(* IEC 61131-3 sources: LTL-Test-Case-Generation/ (part 2) *)

END_FUNCTION_BLOCK

(* ---- SF_EnableSwitch2.st ---- *)
FUNCTION_BLOCK SF_EnableSwitch2
VAR_INPUT
    Activate: BOOL;
    S_SafetyActive: BOOL;
    S_EnableIn: BOOL;
    S_AutoReset: BOOL;
    Reset: BOOL;
END_VAR
VAR_OUTPUT
    Ready: BOOL;
    S_EnableSwitchOut: BOOL;
    SafetyDemand: BOOL;
    ResetRequest: BOOL;
    Error: BOOL;
    DiagCode: UINT;
END_VAR
VAR
    Reset_Before: BOOL;
END_VAR

BEGIN
// state changes

IF NOT Activate THEN
    DiagCode := 16#0000;

    Ready := FALSE;
    S_EnableSwitchOut := FALSE;
    SafetyDemand := FALSE;
    ResetRequest := FALSE;
    Error := FALSE;
    Reset_Before := FALSE;

ELSE
    IF NOT S_SafetyActive THEN
        DiagCode := 16#8002;
    ELSE
        CASE DiagCode OF
        16#0000:
            DiagCode := 16#8002;
        16#8002:
            IF (S_SafetyActive) THEN
                DiagCode := 16#8004;
            END_IF;
        16#8004:
            IF S_EnableIn THEN
                DiagCode := 16#C010;
            ELSE
                DiagCode := 16#8802;
            END_IF;
        16#8802:
            IF S_EnableIn THEN
                DiagCode := 16#8000;
            END_IF;
        16#8000:
            IF NOT S_EnableIn THEN
                DiagCode := 16#8802;
            END_IF;

        16#C010:
            IF Reset AND Reset_Before THEN
                DiagCode := 16#C011;
            ELSIF NOT S_EnableIn AND Reset AND NOT Reset_Before THEN
                DiagCode := 16#8802;
            ELSIF NOT S_EnableIn THEN
                DiagCode := 16#C410;
            END_IF;
        16#C410:
            IF Reset AND Reset_Before THEN
                DiagCode := 16#C011;
            ELSIF NOT S_EnableIn AND Reset AND NOT Reset_Before THEN
                DiagCode := 16#8802;
            ELSIF S_EnableIn THEN
                DiagCode := 16#C010;
            END_IF;
        16#C011:
            IF NOT Reset THEN
                IF S_EnableIn THEN
                    DiagCode := 16#C010;
                ELSE
                    DiagCode := 16#C410;
                END_IF;
            END_IF;
        END_CASE;
    END_IF;

    // set output variables
    CASE DiagCode OF
    16#8002:
        Ready := TRUE;
        S_EnableSwitchOut := FALSE;
        SafetyDemand := FALSE;
        ResetRequest := FALSE;
        Error := FALSE;
    16#8004:
        Ready := TRUE;
        S_EnableSwitchOut := FALSE;
        SafetyDemand := FALSE;
        ResetRequest := FALSE;
        Error := FALSE;
    16#8802:
        Ready := TRUE;
        S_EnableSwitchOut := FALSE;
        SafetyDemand := TRUE;
        ResetRequest := FALSE;
        Error := FALSE;
    16#8000:
        Ready := TRUE;
        S_EnableSwitchOut := TRUE;
        SafetyDemand := FALSE;
        ResetRequest := FALSE;
        Error := FALSE;

    // errors
    16#C011:
        Ready := TRUE;
        S_EnableSwitchOut := FALSE;
        SafetyDemand := FALSE;
        ResetRequest := FALSE;
        Error := TRUE;
    16#C010:
        Ready := TRUE;
        S_EnableSwitchOut := FALSE;
        SafetyDemand := FALSE;
        ResetRequest := FALSE;
        Error := TRUE;
    16#C410:
        Ready := TRUE;
        S_EnableSwitchOut := FALSE;
        SafetyDemand := FALSE;
        ResetRequest := NOT Reset;
        Error := TRUE;
    END_CASE;

    Reset_Before := Reset;
END_IF;

END_FUNCTION_BLOCK

(* ---- SF_EnableSwitch2_Test.st ---- *)
FUNCTION_BLOCK SF_EnableSwitch2_Test
VAR_INPUT
END_VAR
VAR_OUTPUT
	failed_0: BOOL := FALSE;
	finished_0: BOOL := FALSE;
END_VAR
VAR
	fb_0: SF_EnableSwitch2_BranchCounters;
	waitCounter_0: UINT := 0;
	testState_0: UINT := 0;
END_VAR

IF NOT failed_0 AND NOT finished_0 THEN
CASE testState_0 OF
0:
	fb_0.Activate := FALSE; fb_0.S_SafetyActive := FALSE; fb_0.S_EnableIn := FALSE; fb_0.Reset := FALSE;
	fb_0();
	failed_0 := NOT (((((((NOT (fb_0.Ready) AND NOT (fb_0.S_EnableSwitchOut)) AND NOT (fb_0.SafetyDemand)) AND NOT (fb_0.ResetRequest)) AND NOT (fb_0.Error)) AND (fb_0.DiagCode = 0)) AND NOT (fb_0.Reset_Before)));
	testState_0 := testState_0 + 1;
1:
	fb_0.Activate := TRUE; fb_0.S_SafetyActive := FALSE; fb_0.S_EnableIn := FALSE; fb_0.Reset := FALSE;
	fb_0();
	failed_0 := NOT (((((((fb_0.Ready AND NOT (fb_0.S_EnableSwitchOut)) AND NOT (fb_0.SafetyDemand)) AND NOT (fb_0.ResetRequest)) AND NOT (fb_0.Error)) AND (fb_0.DiagCode = 32770)) AND NOT (fb_0.Reset_Before)));
	testState_0 := testState_0 + 1;
2:
	fb_0.Activate := TRUE; fb_0.S_SafetyActive := FALSE; fb_0.S_EnableIn := FALSE; fb_0.Reset := FALSE;
	fb_0();
	failed_0 := NOT (((((((fb_0.Ready AND NOT (fb_0.S_EnableSwitchOut)) AND NOT (fb_0.SafetyDemand)) AND NOT (fb_0.ResetRequest)) AND NOT (fb_0.Error)) AND (fb_0.DiagCode = 32770)) AND NOT (fb_0.Reset_Before)));
	testState_0 := testState_0 + 1;
3:
	fb_0.Activate := TRUE; fb_0.S_SafetyActive := TRUE; fb_0.S_EnableIn := FALSE; fb_0.Reset := FALSE;
	fb_0();
	failed_0 := NOT (((((((fb_0.Ready AND NOT (fb_0.S_EnableSwitchOut)) AND NOT (fb_0.SafetyDemand)) AND NOT (fb_0.ResetRequest)) AND NOT (fb_0.Error)) AND (fb_0.DiagCode = 32772)) AND NOT (fb_0.Reset_Before)));
	testState_0 := testState_0 + 1;
4:
	fb_0.Activate := TRUE; fb_0.S_SafetyActive := TRUE; fb_0.S_EnableIn := FALSE; fb_0.Reset := FALSE;
	fb_0();
	failed_0 := NOT (((((((fb_0.Ready AND NOT (fb_0.S_EnableSwitchOut)) AND fb_0.SafetyDemand) AND NOT (fb_0.ResetRequest)) AND NOT (fb_0.Error)) AND (fb_0.DiagCode = 34818)) AND NOT (fb_0.Reset_Before)));
	testState_0 := testState_0 + 1;
5:
	fb_0.Activate := TRUE; fb_0.S_SafetyActive := TRUE; fb_0.S_EnableIn := FALSE; fb_0.Reset := FALSE;
	fb_0();
	failed_0 := NOT (((((((fb_0.Ready AND NOT (fb_0.S_EnableSwitchOut)) AND fb_0.SafetyDemand) AND NOT (fb_0.ResetRequest)) AND NOT (fb_0.Error)) AND (fb_0.DiagCode = 34818)) AND NOT (fb_0.Reset_Before)));
	testState_0 := testState_0 + 1;
6:
	fb_0.Activate := TRUE; fb_0.S_SafetyActive := TRUE; fb_0.S_EnableIn := TRUE; fb_0.Reset := FALSE;
	fb_0();
	failed_0 := NOT (((((((fb_0.Ready AND fb_0.S_EnableSwitchOut) AND NOT (fb_0.SafetyDemand)) AND NOT (fb_0.ResetRequest)) AND NOT (fb_0.Error)) AND (fb_0.DiagCode = 32768)) AND NOT (fb_0.Reset_Before)));
	testState_0 := testState_0 + 1;
7:
	fb_0.Activate := TRUE; fb_0.S_SafetyActive := TRUE; fb_0.S_EnableIn := TRUE; fb_0.Reset := FALSE;
	fb_0();
	failed_0 := NOT (((((((fb_0.Ready AND fb_0.S_EnableSwitchOut) AND NOT (fb_0.SafetyDemand)) AND NOT (fb_0.ResetRequest)) AND NOT (fb_0.Error)) AND (fb_0.DiagCode = 32768)) AND NOT (fb_0.Reset_Before)));
	testState_0 := testState_0 + 1;
8:
	fb_0.Activate := TRUE; fb_0.S_SafetyActive := TRUE; fb_0.S_EnableIn := FALSE; fb_0.Reset := FALSE;
	fb_0();
	failed_0 := NOT (((((((fb_0.Ready AND NOT (fb_0.S_EnableSwitchOut)) AND fb_0.SafetyDemand) AND NOT (fb_0.ResetRequest)) AND NOT (fb_0.Error)) AND (fb_0.DiagCode = 34818)) AND NOT (fb_0.Reset_Before)));
	testState_0 := testState_0 + 1;
9:
	fb_0.Activate := TRUE; fb_0.S_SafetyActive := FALSE; fb_0.S_EnableIn := FALSE; fb_0.Reset := FALSE;
	fb_0();
	failed_0 := NOT (((((((fb_0.Ready AND NOT (fb_0.S_EnableSwitchOut)) AND NOT (fb_0.SafetyDemand)) AND NOT (fb_0.ResetRequest)) AND NOT (fb_0.Error)) AND (fb_0.DiagCode = 32770)) AND NOT (fb_0.Reset_Before)));
	testState_0 := testState_0 + 1;
10:
	fb_0.Activate := TRUE; fb_0.S_SafetyActive := TRUE; fb_0.S_EnableIn := FALSE; fb_0.Reset := FALSE;
	fb_0();
	failed_0 := NOT (((((((fb_0.Ready AND NOT (fb_0.S_EnableSwitchOut)) AND NOT (fb_0.SafetyDemand)) AND NOT (fb_0.ResetRequest)) AND NOT (fb_0.Error)) AND (fb_0.DiagCode = 32772)) AND NOT (fb_0.Reset_Before)));
	testState_0 := testState_0 + 1;
11:
	fb_0.Activate := TRUE; fb_0.S_SafetyActive := TRUE; fb_0.S_EnableIn := TRUE; fb_0.Reset := TRUE;
	fb_0();
	failed_0 := NOT (((((((fb_0.Ready AND NOT (fb_0.S_EnableSwitchOut)) AND NOT (fb_0.SafetyDemand)) AND NOT (fb_0.ResetRequest)) AND fb_0.Error) AND (fb_0.DiagCode = 49168)) AND fb_0.Reset_Before));
	testState_0 := testState_0 + 1;
12:
	fb_0.Activate := TRUE; fb_0.S_SafetyActive := TRUE; fb_0.S_EnableIn := TRUE; fb_0.Reset := TRUE;
	fb_0();
	failed_0 := NOT (((((((fb_0.Ready AND NOT (fb_0.S_EnableSwitchOut)) AND NOT (fb_0.SafetyDemand)) AND NOT (fb_0.ResetRequest)) AND fb_0.Error) AND (fb_0.DiagCode = 49169)) AND fb_0.Reset_Before));
	testState_0 := testState_0 + 1;
13:
	fb_0.Activate := TRUE; fb_0.S_SafetyActive := TRUE; fb_0.S_EnableIn := TRUE; fb_0.Reset := TRUE;
	fb_0();
	failed_0 := NOT (((((((fb_0.Ready AND NOT (fb_0.S_EnableSwitchOut)) AND NOT (fb_0.SafetyDemand)) AND NOT (fb_0.ResetRequest)) AND fb_0.Error) AND (fb_0.DiagCode = 49169)) AND fb_0.Reset_Before));
	testState_0 := testState_0 + 1;
14:
	fb_0.Activate := TRUE; fb_0.S_SafetyActive := TRUE; fb_0.S_EnableIn := TRUE; fb_0.Reset := FALSE;
	fb_0();
	failed_0 := NOT (((((((fb_0.Ready AND NOT (fb_0.S_EnableSwitchOut)) AND NOT (fb_0.SafetyDemand)) AND NOT (fb_0.ResetRequest)) AND fb_0.Error) AND (fb_0.DiagCode = 49168)) AND NOT (fb_0.Reset_Before)));
	testState_0 := testState_0 + 1;
15:
	fb_0.Activate := TRUE; fb_0.S_SafetyActive := TRUE; fb_0.S_EnableIn := TRUE; fb_0.Reset := FALSE;
	fb_0();
	failed_0 := NOT (((((((fb_0.Ready AND NOT (fb_0.S_EnableSwitchOut)) AND NOT (fb_0.SafetyDemand)) AND NOT (fb_0.ResetRequest)) AND fb_0.Error) AND (fb_0.DiagCode = 49168)) AND NOT (fb_0.Reset_Before)));
	testState_0 := testState_0 + 1;
16:
	fb_0.Activate := TRUE; fb_0.S_SafetyActive := TRUE; fb_0.S_EnableIn := FALSE; fb_0.Reset := FALSE;
	fb_0();
	failed_0 := NOT (((((((fb_0.Ready AND NOT (fb_0.S_EnableSwitchOut)) AND NOT (fb_0.SafetyDemand)) AND fb_0.ResetRequest) AND fb_0.Error) AND (fb_0.DiagCode = 50192)) AND NOT (fb_0.Reset_Before)));
	testState_0 := testState_0 + 1;
17:
	fb_0.Activate := TRUE; fb_0.S_SafetyActive := TRUE; fb_0.S_EnableIn := FALSE; fb_0.Reset := FALSE;
	fb_0();
	failed_0 := NOT (((((((fb_0.Ready AND NOT (fb_0.S_EnableSwitchOut)) AND NOT (fb_0.SafetyDemand)) AND fb_0.ResetRequest) AND fb_0.Error) AND (fb_0.DiagCode = 50192)) AND NOT (fb_0.Reset_Before)));
	testState_0 := testState_0 + 1;
18:
	fb_0.Activate := TRUE; fb_0.S_SafetyActive := TRUE; fb_0.S_EnableIn := TRUE; fb_0.Reset := FALSE;
	fb_0();
	failed_0 := NOT (((((((fb_0.Ready AND NOT (fb_0.S_EnableSwitchOut)) AND NOT (fb_0.SafetyDemand)) AND NOT (fb_0.ResetRequest)) AND fb_0.Error) AND (fb_0.DiagCode = 49168)) AND NOT (fb_0.Reset_Before)));
	testState_0 := testState_0 + 1;
19:
	fb_0.Activate := TRUE; fb_0.S_SafetyActive := TRUE; fb_0.S_EnableIn := FALSE; fb_0.Reset := TRUE;
	fb_0();
	failed_0 := NOT (((((((fb_0.Ready AND NOT (fb_0.S_EnableSwitchOut)) AND fb_0.SafetyDemand) AND NOT (fb_0.ResetRequest)) AND NOT (fb_0.Error)) AND (fb_0.DiagCode = 34818)) AND fb_0.Reset_Before));
	testState_0 := testState_0 + 1;
20:
	fb_0.Activate := TRUE; fb_0.S_SafetyActive := FALSE; fb_0.S_EnableIn := FALSE; fb_0.Reset := FALSE;
	fb_0();
	failed_0 := NOT (((((((fb_0.Ready AND NOT (fb_0.S_EnableSwitchOut)) AND NOT (fb_0.SafetyDemand)) AND NOT (fb_0.ResetRequest)) AND NOT (fb_0.Error)) AND (fb_0.DiagCode = 32770)) AND NOT (fb_0.Reset_Before)));
	testState_0 := testState_0 + 1;
21:
	fb_0.Activate := TRUE; fb_0.S_SafetyActive := FALSE; fb_0.S_EnableIn := FALSE; fb_0.Reset := FALSE;
	fb_0();
	failed_0 := NOT (((((((fb_0.Ready AND NOT (fb_0.S_EnableSwitchOut)) AND NOT (fb_0.SafetyDemand)) AND NOT (fb_0.ResetRequest)) AND NOT (fb_0.Error)) AND (fb_0.DiagCode = 32770)) AND NOT (fb_0.Reset_Before)));
	testState_0 := testState_0 + 1;
22:
	fb_0.Activate := TRUE; fb_0.S_SafetyActive := TRUE; fb_0.S_EnableIn := FALSE; fb_0.Reset := FALSE;
	fb_0();
	failed_0 := NOT (((((((fb_0.Ready AND NOT (fb_0.S_EnableSwitchOut)) AND NOT (fb_0.SafetyDemand)) AND NOT (fb_0.ResetRequest)) AND NOT (fb_0.Error)) AND (fb_0.DiagCode = 32772)) AND NOT (fb_0.Reset_Before)));
	testState_0 := testState_0 + 1;
23:
	fb_0.Activate := TRUE; fb_0.S_SafetyActive := TRUE; fb_0.S_EnableIn := TRUE; fb_0.Reset := TRUE;
	fb_0();
	failed_0 := NOT (((((((fb_0.Ready AND NOT (fb_0.S_EnableSwitchOut)) AND NOT (fb_0.SafetyDemand)) AND NOT (fb_0.ResetRequest)) AND fb_0.Error) AND (fb_0.DiagCode = 49168)) AND fb_0.Reset_Before));
	testState_0 := testState_0 + 1;
24:
	fb_0.Activate := TRUE; fb_0.S_SafetyActive := TRUE; fb_0.S_EnableIn := FALSE; fb_0.Reset := TRUE;
	fb_0();
	failed_0 := NOT (((((((fb_0.Ready AND NOT (fb_0.S_EnableSwitchOut)) AND NOT (fb_0.SafetyDemand)) AND NOT (fb_0.ResetRequest)) AND fb_0.Error) AND (fb_0.DiagCode = 49169)) AND fb_0.Reset_Before));
	testState_0 := testState_0 + 1;
25:
	fb_0.Activate := TRUE; fb_0.S_SafetyActive := TRUE; fb_0.S_EnableIn := FALSE; fb_0.Reset := FALSE;
	fb_0();
	failed_0 := NOT (((((((fb_0.Ready AND NOT (fb_0.S_EnableSwitchOut)) AND NOT (fb_0.SafetyDemand)) AND fb_0.ResetRequest) AND fb_0.Error) AND (fb_0.DiagCode = 50192)) AND NOT (fb_0.Reset_Before)));
	testState_0 := testState_0 + 1;
26:
	fb_0.Activate := TRUE; fb_0.S_SafetyActive := TRUE; fb_0.S_EnableIn := FALSE; fb_0.Reset := TRUE;
	fb_0();
	failed_0 := NOT (((((((fb_0.Ready AND NOT (fb_0.S_EnableSwitchOut)) AND fb_0.SafetyDemand) AND NOT (fb_0.ResetRequest)) AND NOT (fb_0.Error)) AND (fb_0.DiagCode = 34818)) AND fb_0.Reset_Before));
	testState_0 := testState_0 + 1;
27:
	fb_0.Activate := TRUE; fb_0.S_SafetyActive := FALSE; fb_0.S_EnableIn := FALSE; fb_0.Reset := FALSE;
	fb_0();
	failed_0 := NOT ((fb_0.Ready AND (NOT (fb_0.S_EnableSwitchOut) AND (NOT (fb_0.SafetyDemand) AND (NOT (fb_0.ResetRequest) AND (NOT (fb_0.Error) AND ((fb_0.DiagCode = 32770) AND NOT (fb_0.Reset_Before))))))));
	testState_0 := testState_0 + 1;
28:
	finished_0 := TRUE;
END_CASE
END_IF

END_FUNCTION_BLOCK

(* ---- SF_Equivalent_U.st ---- *)
FUNCTION_BLOCK SF_Equivalent_U
VAR_INPUT
    Activate: BOOL;
    S_ChannelA: BOOL;
    S_ChannelB: BOOL;
    DiscrepancyTime: TIME := T#100ms;
END_VAR
VAR_OUTPUT
    Ready: BOOL;
    S_EquivalentOut: BOOL;
    SafetyDemand: BOOL;
    Error: BOOL;
    DiagCode: UINT;
END_VAR
VAR
    T_1: TON;
END_VAR

BEGIN

// state changes
IF NOT Activate THEN
    DiagCode := 16#0000;
    T_1(IN := 0);

    Ready := FALSE;
    SafetyDemand := FALSE;
    Error := FALSE;
    S_EquivalentOut := FALSE;
ELSE
    T_1(PT := DiscrepancyTime);

    CASE DiagCode OF
    16#0000:
        DiagCode := 16#8801;
    16#8000:
        IF S_ChannelA XOR S_ChannelB THEN
            DiagCode := 16#8806;
            T_1(IN := 0);
            T_1(IN := 1, PT := DiscrepancyTime);
        ELSIF NOT S_ChannelA AND NOT S_ChannelB THEN
            T_1(IN := 0);
            DiagCode := 16#8801;
        END_IF;
    16#8801:
        IF S_ChannelA AND NOT S_ChannelB THEN
            DiagCode := 16#8802;
            T_1(IN := 0);
            T_1(IN := 1, PT := DiscrepancyTime);
        ELSIF S_ChannelB AND NOT S_ChannelA THEN
            DiagCode := 16#8804;
            T_1(IN := 0);
            T_1(IN := 1, PT := DiscrepancyTime);
        ELSIF S_ChannelA AND S_ChannelB THEN
            DiagCode := 16#8000;
        END_IF;
    16#8802:
        IF T_1.Q THEN
            DiagCode := 16#C010;
        ELSIF NOT S_ChannelA THEN
            T_1(IN := 0);
            DiagCode := 16#8801;
        ELSIF S_ChannelB THEN
            T_1(IN := 0);
            DiagCode := 16#8000;
        END_IF;
    16#8804:
        IF T_1.Q THEN
            DiagCode := 16#C020;
        ELSIF NOT S_ChannelB THEN
            T_1(IN := 0);
            DiagCode := 16#8801;
        ELSIF S_ChannelA THEN
            T_1(IN := 0);
            DiagCode := 16#8000;
        END_IF;
    16#8806:
        IF T_1.Q THEN
            DiagCode := 16#C030;
        ELSIF NOT S_ChannelA AND NOT S_ChannelB THEN
            T_1(IN := 0);
            DiagCode := 16#8801;
        END_IF;
    16#C010:
        IF NOT S_ChannelA AND NOT S_ChannelB THEN
            T_1(IN := 0);
            DiagCode := 16#8801;
        END_IF;
    16#C020:
        IF NOT S_ChannelA AND NOT S_ChannelB THEN
            T_1(IN := 0);
            DiagCode := 16#8801;
        END_IF;
    16#C030:
        IF NOT S_ChannelA AND NOT S_ChannelB THEN
            T_1(IN := 0);
            DiagCode := 16#8801;
        END_IF;
    END_CASE;

    // set output variables
    CASE DiagCode OF
    16#8000:
        Ready := TRUE;
        SafetyDemand := FALSE;
        Error := FALSE;
        S_EquivalentOut := TRUE;
    16#8801:
        Ready := TRUE;
        SafetyDemand := TRUE;
        Error := FALSE;
        S_EquivalentOut := FALSE;
    16#8802:
        Ready := TRUE;
        SafetyDemand := TRUE;
        Error := FALSE;
        S_EquivalentOut := FALSE;
    16#8804:
        Ready := TRUE;
        SafetyDemand := TRUE;
        Error := FALSE;
        S_EquivalentOut := FALSE;
    16#8806:
        Ready := TRUE;
        SafetyDemand := TRUE;
        Error := FALSE;
        S_EquivalentOut := FALSE;
    16#C010:
        Ready := TRUE;
        SafetyDemand := FALSE;
        Error := TRUE;
        S_EquivalentOut := FALSE;
    16#C020:
        Ready := TRUE;
        SafetyDemand := FALSE;
        Error := TRUE;
        S_EquivalentOut := FALSE;
    16#C030:
        Ready := TRUE;
        SafetyDemand := FALSE;
        Error := TRUE;
        S_EquivalentOut := FALSE;
    END_CASE;
END_IF;

END_FUNCTION_BLOCK

(* ---- SF_Equivalent_U_Test.st ---- *)
FUNCTION_BLOCK SF_Equivalent_U_Test
VAR_INPUT
END_VAR
VAR_OUTPUT
	failed_0: BOOL := FALSE;
	finished_0: BOOL := FALSE;
END_VAR
VAR
	fb_0: SF_Equivalent_U_BranchCounters;
	waitCounter_0: UINT := 0;
	testState_0: UINT := 0;
END_VAR

IF NOT failed_0 AND NOT finished_0 THEN
CASE testState_0 OF
0:
	fb_0.Activate := FALSE;
	fb_0();
	failed_0 := NOT ((((((NOT (fb_0.T_1.Q) AND (fb_0.DiagCode = 0)) AND NOT (fb_0.Ready)) AND NOT (fb_0.S_EquivalentOut)) AND NOT (fb_0.SafetyDemand)) AND NOT (fb_0.Error)));
	testState_0 := testState_0 + 1;
1:
	fb_0.Activate := TRUE; fb_0.S_ChannelA := FALSE; fb_0.S_ChannelB := FALSE;
	fb_0();
	failed_0 := NOT ((((((NOT (fb_0.T_1.Q) AND (fb_0.DiagCode = 34817)) AND fb_0.Ready) AND NOT (fb_0.S_EquivalentOut)) AND fb_0.SafetyDemand) AND NOT (fb_0.Error)));
	testState_0 := testState_0 + 1;
2:
	fb_0.Activate := TRUE; fb_0.S_ChannelA := FALSE; fb_0.S_ChannelB := FALSE;
	fb_0();
	failed_0 := NOT ((((((NOT (fb_0.T_1.Q) AND (fb_0.DiagCode = 34817)) AND fb_0.Ready) AND NOT (fb_0.S_EquivalentOut)) AND fb_0.SafetyDemand) AND NOT (fb_0.Error)));
	testState_0 := testState_0 + 1;
3:
	fb_0.Activate := TRUE; fb_0.S_ChannelA := TRUE; fb_0.S_ChannelB := FALSE;
	fb_0();
	failed_0 := NOT ((((((NOT (fb_0.T_1.Q) AND (fb_0.DiagCode = 34818)) AND fb_0.Ready) AND NOT (fb_0.S_EquivalentOut)) AND fb_0.SafetyDemand) AND NOT (fb_0.Error)));
	testState_0 := testState_0 + 1;
4:
	fb_0.Activate := TRUE; fb_0.S_ChannelA := FALSE; fb_0.S_ChannelB := FALSE;
	fb_0();
	IF fb_0.T_1.Q THEN
		finished_0 := TRUE;
	ELSE
		testState_0 := testState_0 + 1;
	END_IF
5:
	failed_0 := NOT ((((((NOT (fb_0.T_1.Q) AND (fb_0.DiagCode = 34817)) AND fb_0.Ready) AND NOT (fb_0.S_EquivalentOut)) AND fb_0.SafetyDemand) AND NOT (fb_0.Error)));
	testState_0 := testState_0 + 1;
6:
	fb_0.Activate := TRUE; fb_0.S_ChannelA := TRUE; fb_0.S_ChannelB := FALSE;
	fb_0();
	failed_0 := NOT ((((((NOT (fb_0.T_1.Q) AND (fb_0.DiagCode = 34818)) AND fb_0.Ready) AND NOT (fb_0.S_EquivalentOut)) AND fb_0.SafetyDemand) AND NOT (fb_0.Error)));
	testState_0 := testState_0 + 1;
7:
	fb_0.Activate := TRUE; fb_0.S_ChannelA := TRUE; fb_0.S_ChannelB := TRUE;
	fb_0();
	IF fb_0.T_1.Q THEN
		finished_0 := TRUE;
	ELSE
		testState_0 := testState_0 + 1;
	END_IF
8:
	failed_0 := NOT ((((((NOT (fb_0.T_1.Q) AND (fb_0.DiagCode = 32768)) AND fb_0.Ready) AND fb_0.S_EquivalentOut) AND NOT (fb_0.SafetyDemand)) AND NOT (fb_0.Error)));
	testState_0 := testState_0 + 1;
9:
	fb_0.Activate := TRUE; fb_0.S_ChannelA := TRUE; fb_0.S_ChannelB := TRUE;
	fb_0();
	failed_0 := NOT ((((((NOT (fb_0.T_1.Q) AND (fb_0.DiagCode = 32768)) AND fb_0.Ready) AND fb_0.S_EquivalentOut) AND NOT (fb_0.SafetyDemand)) AND NOT (fb_0.Error)));
	testState_0 := testState_0 + 1;
10:
	fb_0.Activate := TRUE; fb_0.S_ChannelA := FALSE; fb_0.S_ChannelB := TRUE;
	fb_0();
	failed_0 := NOT ((((((NOT (fb_0.T_1.Q) AND (fb_0.DiagCode = 34822)) AND fb_0.Ready) AND NOT (fb_0.S_EquivalentOut)) AND fb_0.SafetyDemand) AND NOT (fb_0.Error)));
	testState_0 := testState_0 + 1;
11:
	fb_0.Activate := TRUE; fb_0.S_ChannelA := FALSE; fb_0.S_ChannelB := FALSE;
	fb_0();
	IF fb_0.T_1.Q THEN
		finished_0 := TRUE;
	ELSE
		testState_0 := testState_0 + 1;
	END_IF
12:
	failed_0 := NOT ((((((NOT (fb_0.T_1.Q) AND (fb_0.DiagCode = 34817)) AND fb_0.Ready) AND NOT (fb_0.S_EquivalentOut)) AND fb_0.SafetyDemand) AND NOT (fb_0.Error)));
	testState_0 := testState_0 + 1;
13:
	fb_0.Activate := TRUE; fb_0.S_ChannelA := FALSE; fb_0.S_ChannelB := TRUE;
	fb_0();
	failed_0 := NOT ((((((NOT (fb_0.T_1.Q) AND (fb_0.DiagCode = 34820)) AND fb_0.Ready) AND NOT (fb_0.S_EquivalentOut)) AND fb_0.SafetyDemand) AND NOT (fb_0.Error)));
	testState_0 := testState_0 + 1;
14:
	fb_0.Activate := TRUE; fb_0.S_ChannelA := FALSE; fb_0.S_ChannelB := FALSE;
	fb_0();
	IF fb_0.T_1.Q THEN
		finished_0 := TRUE;
	ELSE
		testState_0 := testState_0 + 1;
	END_IF
15:
	failed_0 := NOT ((((((NOT (fb_0.T_1.Q) AND (fb_0.DiagCode = 34817)) AND fb_0.Ready) AND NOT (fb_0.S_EquivalentOut)) AND fb_0.SafetyDemand) AND NOT (fb_0.Error)));
	testState_0 := testState_0 + 1;
16:
	fb_0.Activate := TRUE; fb_0.S_ChannelA := FALSE; fb_0.S_ChannelB := TRUE;
	fb_0();
	failed_0 := NOT ((((((NOT (fb_0.T_1.Q) AND (fb_0.DiagCode = 34820)) AND fb_0.Ready) AND NOT (fb_0.S_EquivalentOut)) AND fb_0.SafetyDemand) AND NOT (fb_0.Error)));
	testState_0 := testState_0 + 1;
17:
	fb_0.Activate := TRUE; fb_0.S_ChannelA := TRUE; fb_0.S_ChannelB := TRUE;
	fb_0();
	IF fb_0.T_1.Q THEN
		finished_0 := TRUE;
	ELSE
		testState_0 := testState_0 + 1;
	END_IF
18:
	failed_0 := NOT ((((((NOT (fb_0.T_1.Q) AND (fb_0.DiagCode = 32768)) AND fb_0.Ready) AND fb_0.S_EquivalentOut) AND NOT (fb_0.SafetyDemand)) AND NOT (fb_0.Error)));
	testState_0 := testState_0 + 1;
19:
	fb_0.Activate := TRUE; fb_0.S_ChannelA := FALSE; fb_0.S_ChannelB := FALSE;
	fb_0();
	failed_0 := NOT ((((((NOT (fb_0.T_1.Q) AND (fb_0.DiagCode = 34817)) AND fb_0.Ready) AND NOT (fb_0.S_EquivalentOut)) AND fb_0.SafetyDemand) AND NOT (fb_0.Error)));
	testState_0 := testState_0 + 1;
20:
	fb_0.Activate := TRUE; fb_0.S_ChannelA := TRUE; fb_0.S_ChannelB := TRUE;
	fb_0();
	failed_0 := NOT ((((((NOT (fb_0.T_1.Q) AND (fb_0.DiagCode = 32768)) AND fb_0.Ready) AND fb_0.S_EquivalentOut) AND NOT (fb_0.SafetyDemand)) AND NOT (fb_0.Error)));
	testState_0 := testState_0 + 1;
21:
	fb_0.Activate := TRUE; fb_0.S_ChannelA := TRUE; fb_0.S_ChannelB := FALSE;
	fb_0();
	failed_0 := NOT ((((((NOT (fb_0.T_1.Q) AND (fb_0.DiagCode = 34822)) AND fb_0.Ready) AND NOT (fb_0.S_EquivalentOut)) AND fb_0.SafetyDemand) AND NOT (fb_0.Error)));
	testState_0 := testState_0 + 1;
22:
	IF (fb_0.T_1.Q AND (fb_0.DiagCode = 49200)) THEN
		waitCounter_0 := 0;
		testState_0 := testState_0 + 1;
	ELSE
		failed_0 := NOT ((NOT (fb_0.T_1.Q) AND ((fb_0.DiagCode = 34822) AND (fb_0.Ready AND (NOT (fb_0.S_EquivalentOut) AND (fb_0.SafetyDemand AND NOT (fb_0.Error)))))));
		IF waitCounter_0 > 100 THEN
			finished_0 := TRUE;
		ELSE
			waitCounter_0 := waitCounter_0 + 1;
			fb_0();
		END_IF
	END_IF
23:
	failed_0 := NOT ((((((fb_0.T_1.Q AND (fb_0.DiagCode = 49200)) AND fb_0.Ready) AND NOT (fb_0.S_EquivalentOut)) AND NOT (fb_0.SafetyDemand)) AND fb_0.Error));
	testState_0 := testState_0 + 1;
24:
	fb_0.Activate := TRUE; fb_0.S_ChannelA := TRUE; fb_0.S_ChannelB := FALSE;
	fb_0();
	failed_0 := NOT ((((((fb_0.T_1.Q AND (fb_0.DiagCode = 49200)) AND fb_0.Ready) AND NOT (fb_0.S_EquivalentOut)) AND NOT (fb_0.SafetyDemand)) AND fb_0.Error));
	testState_0 := testState_0 + 1;
25:
	fb_0.Activate := TRUE; fb_0.S_ChannelA := FALSE; fb_0.S_ChannelB := FALSE;
	fb_0();
	failed_0 := NOT ((((((NOT (fb_0.T_1.Q) AND (fb_0.DiagCode = 34817)) AND fb_0.Ready) AND NOT (fb_0.S_EquivalentOut)) AND fb_0.SafetyDemand) AND NOT (fb_0.Error)));
	testState_0 := testState_0 + 1;
26:
	fb_0.Activate := TRUE; fb_0.S_ChannelA := TRUE; fb_0.S_ChannelB := FALSE;
	fb_0();
	failed_0 := NOT ((((((NOT (fb_0.T_1.Q) AND (fb_0.DiagCode = 34818)) AND fb_0.Ready) AND NOT (fb_0.S_EquivalentOut)) AND fb_0.SafetyDemand) AND NOT (fb_0.Error)));
	testState_0 := testState_0 + 1;
27:
	IF (fb_0.T_1.Q AND (fb_0.DiagCode = 49168)) THEN
		waitCounter_0 := 0;
		testState_0 := testState_0 + 1;
	ELSE
		failed_0 := NOT ((NOT (fb_0.T_1.Q) AND ((fb_0.DiagCode = 34818) AND (fb_0.Ready AND (NOT (fb_0.S_EquivalentOut) AND (fb_0.SafetyDemand AND NOT (fb_0.Error)))))));
		IF waitCounter_0 > 100 THEN
			finished_0 := TRUE;
		ELSE
			waitCounter_0 := waitCounter_0 + 1;
			fb_0();
		END_IF
	END_IF
28:
	failed_0 := NOT ((((((fb_0.T_1.Q AND (fb_0.DiagCode = 49168)) AND fb_0.Ready) AND NOT (fb_0.S_EquivalentOut)) AND NOT (fb_0.SafetyDemand)) AND fb_0.Error));
	testState_0 := testState_0 + 1;
29:
	fb_0.Activate := TRUE; fb_0.S_ChannelA := TRUE; fb_0.S_ChannelB := FALSE;
	fb_0();
	failed_0 := NOT ((((((fb_0.T_1.Q AND (fb_0.DiagCode = 49168)) AND fb_0.Ready) AND NOT (fb_0.S_EquivalentOut)) AND NOT (fb_0.SafetyDemand)) AND fb_0.Error));
	testState_0 := testState_0 + 1;
30:
	fb_0.Activate := TRUE; fb_0.S_ChannelA := FALSE; fb_0.S_ChannelB := FALSE;
	fb_0();
	failed_0 := NOT ((((((NOT (fb_0.T_1.Q) AND (fb_0.DiagCode = 34817)) AND fb_0.Ready) AND NOT (fb_0.S_EquivalentOut)) AND fb_0.SafetyDemand) AND NOT (fb_0.Error)));
	testState_0 := testState_0 + 1;
31:
	fb_0.Activate := TRUE; fb_0.S_ChannelA := FALSE; fb_0.S_ChannelB := TRUE;
	fb_0();
	failed_0 := NOT ((((((NOT (fb_0.T_1.Q) AND (fb_0.DiagCode = 34820)) AND fb_0.Ready) AND NOT (fb_0.S_EquivalentOut)) AND fb_0.SafetyDemand) AND NOT (fb_0.Error)));
	testState_0 := testState_0 + 1;
32:
	IF (fb_0.T_1.Q AND (fb_0.DiagCode = 49184)) THEN
		waitCounter_0 := 0;
		testState_0 := testState_0 + 1;
	ELSE
		failed_0 := NOT ((NOT (fb_0.T_1.Q) AND ((fb_0.DiagCode = 34820) AND (fb_0.Ready AND (NOT (fb_0.S_EquivalentOut) AND (fb_0.SafetyDemand AND NOT (fb_0.Error)))))));
		IF waitCounter_0 > 100 THEN
			finished_0 := TRUE;
		ELSE
			waitCounter_0 := waitCounter_0 + 1;
			fb_0();
		END_IF
	END_IF
33:
	failed_0 := NOT ((((((fb_0.T_1.Q AND (fb_0.DiagCode = 49184)) AND fb_0.Ready) AND NOT (fb_0.S_EquivalentOut)) AND NOT (fb_0.SafetyDemand)) AND fb_0.Error));
	testState_0 := testState_0 + 1;
34:
	fb_0.Activate := TRUE; fb_0.S_ChannelA := FALSE; fb_0.S_ChannelB := TRUE;
	fb_0();
	failed_0 := NOT ((((((fb_0.T_1.Q AND (fb_0.DiagCode = 49184)) AND fb_0.Ready) AND NOT (fb_0.S_EquivalentOut)) AND NOT (fb_0.SafetyDemand)) AND fb_0.Error));
	testState_0 := testState_0 + 1;
35:
	fb_0.Activate := TRUE; fb_0.S_ChannelA := FALSE; fb_0.S_ChannelB := FALSE;
	fb_0();
	failed_0 := NOT ((NOT (fb_0.T_1.Q) AND ((fb_0.DiagCode = 34817) AND (fb_0.Ready AND (NOT (fb_0.S_EquivalentOut) AND (fb_0.SafetyDemand AND NOT (fb_0.Error)))))));
	testState_0 := testState_0 + 1;
36:
	finished_0 := TRUE;
END_CASE
END_IF

END_FUNCTION_BLOCK

(* ---- SF_FootSwitch.st ---- *)
FUNCTION_BLOCK SF_FootSwitch
VAR_INPUT
    Activate: BOOL;
    S_SafetyActive: BOOL;
    S_FootSwitchCh1: BOOL;
    S_FootSwitchCh2: BOOL;
    S_AutoReset: BOOL;
    Reset: BOOL;
END_VAR
VAR_OUTPUT
    Ready: BOOL;
    S_FootSwitchOut: BOOL;
    SafetyDemand: BOOL;
    ResetRequest: BOOL;
    Error: BOOL;
    DiagCode: UINT;
END_VAR
VAR
    Reset_Before: BOOL;
    Position1: BOOL;
    Position2: BOOL;
    Position3: BOOL;
END_VAR

BEGIN

IF NOT Activate THEN
    DiagCode := 16#0000;

    Ready := FALSE;
    S_FootSwitchOut := FALSE;
    SafetyDemand := FALSE;
    ResetRequest := FALSE;
    Error := FALSE;
    Reset_Before := FALSE;
    Position1 := FALSE;
    Position2 := FALSE;
    Position3 := FALSE;

ELSE
    // state changes
    IF NOT S_SafetyActive THEN
        DiagCode := 16#8004;

    ELSE
        Position1 := NOT S_FootSwitchCh1 AND S_FootSwitchCh2;
        Position2 := S_FootSwitchCh1 AND S_FootSwitchCh2;
        Position3 := (NOT (S_FootSwitchCh1 OR S_FootSwitchCh2)) OR (S_FootSwitchCh1 AND NOT S_FootSwitchCh2);

        CASE DiagCode OF
        16#0000:
            DiagCode := 16#8004;
        16#8004:
            IF (S_SafetyActive) THEN
                DiagCode := 16#8005;
            END_IF;
        16#8005:
            IF (NOT Position1) THEN
                DiagCode := 16#C120;
            ELSE
                DiagCode := 16#8006;
            END_IF;
        16#8006:
            IF Position2 THEN
                DiagCode := 16#8000;
            ELSIF Position3 THEN
                DiagCode := 16#8810;
            END_IF;
        16#8000:
            IF Position3 THEN
                DiagCode := 16#8810;
            ELSIF Position1 THEN
                DiagCode := 16#8006;
            END_IF;
        16#8810:
            IF Position2 THEN
                DiagCode := 16#C160;
            ELSIF Position1 THEN
                DiagCode := 16#8006;
            END_IF;
        16#C120:
            IF Position1 THEN
                DiagCode := 16#C140;
            END_IF;
        16#C140:
            IF NOT Position1 THEN
                DiagCode := 16#C120;
            ELSIF Reset AND Reset_Before AND NOT S_AutoReset THEN
                DiagCode := 16#C141;
            ELSIF (Reset AND NOT Reset_Before) OR S_AutoReset THEN
                DiagCode := 16#8006;
            END_IF;
        16#C141:
            IF NOT Reset THEN
                DiagCode := 16#C140;
            END_IF;
        16#C160:
            IF NOT Position2 THEN
                DiagCode := 16#C180;
            END_IF;
        16#C180:
            IF Position2 THEN
                DiagCode := 16#C160;
            ELSIF Reset AND Reset_Before AND NOT S_AutoReset THEN
                DiagCode := 16#C181;
            ELSIF (Reset AND NOT Reset_Before) OR S_AutoReset THEN
                DiagCode := 16#8810;
            END_IF;
        16#C181:
            IF NOT Reset THEN
                DiagCode := 16#C180;
            END_IF;
        END_CASE;
    END_IF;

    // set output variables
    CASE DiagCode OF
    16#8004:
        Ready := TRUE;
        S_FootSwitchOut := FALSE;
        SafetyDemand := FALSE;
        ResetRequest := FALSE;
        Error := FALSE;
    16#8005:
        Ready := TRUE;
        S_FootSwitchOut := FALSE;
        SafetyDemand := FALSE;
        ResetRequest := FALSE;
        Error := FALSE;
    16#8006:
        Ready := TRUE;
        S_FootSwitchOut := FALSE;
        SafetyDemand := TRUE;
        ResetRequest := FALSE;
        Error := FALSE;
    16#8810:
        Ready := TRUE;
        S_FootSwitchOut := FALSE;
        SafetyDemand := TRUE;
        ResetRequest := FALSE;
        Error := FALSE;
    16#8000:
        Ready := TRUE;
        S_FootSwitchOut := TRUE;
        SafetyDemand := TRUE;
        ResetRequest := FALSE;
        Error := FALSE;

    // errors
    16#C141:
        Ready := TRUE;
        S_FootSwitchOut := FALSE;
        SafetyDemand := FALSE;
        ResetRequest := FALSE;
        Error := TRUE;
    16#C181:
        Ready := TRUE;
        S_FootSwitchOut := FALSE;
        SafetyDemand := FALSE;
        ResetRequest := FALSE;
        Error := TRUE;
    16#C120:
        Ready := TRUE;
        S_FootSwitchOut := FALSE;
        SafetyDemand := FALSE;
        ResetRequest := FALSE;
        Error := TRUE;
    16#C140:
        Ready := TRUE;
        S_FootSwitchOut := FALSE;
        SafetyDemand := FALSE;
        ResetRequest := FALSE;
        Error := TRUE;
    16#C160:
        Ready := TRUE;
        S_FootSwitchOut := FALSE;
        SafetyDemand := FALSE;
        ResetRequest := FALSE;
        Error := TRUE;
    16#C180:
        Ready := TRUE;
        S_FootSwitchOut := FALSE;
        SafetyDemand := FALSE;
        ResetRequest := FALSE;
        Error := TRUE;
    END_CASE;

    Reset_Before := Reset;
END_IF;

END_FUNCTION_BLOCK

(* ---- SF_FootSwitch_Test.st ---- *)
FUNCTION_BLOCK SF_FootSwitch_Test
VAR_INPUT
END_VAR
VAR_OUTPUT
	failed_0: BOOL := FALSE;
	finished_0: BOOL := FALSE;
END_VAR
VAR
	fb_0: SF_FootSwitch_BranchCounters;
	waitCounter_0: UINT := 0;
	testState_0: UINT := 0;
END_VAR

IF NOT failed_0 AND NOT finished_0 THEN
CASE testState_0 OF
0:
	fb_0.Activate := FALSE; fb_0.S_SafetyActive := FALSE; fb_0.S_FootSwitchCh1 := FALSE; fb_0.S_FootSwitchCh2 := FALSE; fb_0.S_AutoReset := FALSE; fb_0.Reset := FALSE;
	fb_0();
	failed_0 := NOT ((((((((((NOT (fb_0.Ready) AND NOT (fb_0.S_FootSwitchOut)) AND NOT (fb_0.SafetyDemand)) AND NOT (fb_0.ResetRequest)) AND NOT (fb_0.Error)) AND (fb_0.DiagCode = 0)) AND NOT (fb_0.Reset_Before)) AND NOT (fb_0.Position1)) AND NOT (fb_0.Position2)) AND NOT (fb_0.Position3)));
	testState_0 := testState_0 + 1;
1:
	fb_0.Activate := TRUE; fb_0.S_SafetyActive := FALSE; fb_0.S_FootSwitchCh1 := FALSE; fb_0.S_FootSwitchCh2 := TRUE; fb_0.S_AutoReset := FALSE; fb_0.Reset := FALSE;
	fb_0();
	failed_0 := NOT ((((((((((fb_0.Ready AND NOT (fb_0.S_FootSwitchOut)) AND NOT (fb_0.SafetyDemand)) AND NOT (fb_0.ResetRequest)) AND NOT (fb_0.Error)) AND (fb_0.DiagCode = 32772)) AND NOT (fb_0.Reset_Before)) AND NOT (fb_0.Position1)) AND NOT (fb_0.Position2)) AND NOT (fb_0.Position3)));
	testState_0 := testState_0 + 1;
2:
	fb_0.Activate := TRUE; fb_0.S_SafetyActive := FALSE; fb_0.S_FootSwitchCh1 := FALSE; fb_0.S_FootSwitchCh2 := TRUE; fb_0.S_AutoReset := FALSE; fb_0.Reset := FALSE;
	fb_0();
	failed_0 := NOT ((((((((((fb_0.Ready AND NOT (fb_0.S_FootSwitchOut)) AND NOT (fb_0.SafetyDemand)) AND NOT (fb_0.ResetRequest)) AND NOT (fb_0.Error)) AND (fb_0.DiagCode = 32772)) AND NOT (fb_0.Reset_Before)) AND NOT (fb_0.Position1)) AND NOT (fb_0.Position2)) AND NOT (fb_0.Position3)));
	testState_0 := testState_0 + 1;
3:
	fb_0.Activate := TRUE; fb_0.S_SafetyActive := TRUE; fb_0.S_FootSwitchCh1 := FALSE; fb_0.S_FootSwitchCh2 := TRUE; fb_0.S_AutoReset := FALSE; fb_0.Reset := FALSE;
	fb_0();
	failed_0 := NOT ((((((((((fb_0.Ready AND NOT (fb_0.S_FootSwitchOut)) AND NOT (fb_0.SafetyDemand)) AND NOT (fb_0.ResetRequest)) AND NOT (fb_0.Error)) AND (fb_0.DiagCode = 32773)) AND NOT (fb_0.Reset_Before)) AND fb_0.Position1) AND NOT (fb_0.Position2)) AND NOT (fb_0.Position3)));
	testState_0 := testState_0 + 1;
4:
	fb_0.Activate := TRUE; fb_0.S_SafetyActive := TRUE; fb_0.S_FootSwitchCh1 := FALSE; fb_0.S_FootSwitchCh2 := TRUE; fb_0.S_AutoReset := FALSE; fb_0.Reset := FALSE;
	fb_0();
	failed_0 := NOT ((((((((((fb_0.Ready AND NOT (fb_0.S_FootSwitchOut)) AND fb_0.SafetyDemand) AND NOT (fb_0.ResetRequest)) AND NOT (fb_0.Error)) AND (fb_0.DiagCode = 32774)) AND NOT (fb_0.Reset_Before)) AND fb_0.Position1) AND NOT (fb_0.Position2)) AND NOT (fb_0.Position3)));
	testState_0 := testState_0 + 1;
5:
	fb_0.Activate := TRUE; fb_0.S_SafetyActive := TRUE; fb_0.S_FootSwitchCh1 := FALSE; fb_0.S_FootSwitchCh2 := TRUE; fb_0.S_AutoReset := FALSE; fb_0.Reset := FALSE;
	fb_0();
	failed_0 := NOT ((((((((((fb_0.Ready AND NOT (fb_0.S_FootSwitchOut)) AND fb_0.SafetyDemand) AND NOT (fb_0.ResetRequest)) AND NOT (fb_0.Error)) AND (fb_0.DiagCode = 32774)) AND NOT (fb_0.Reset_Before)) AND fb_0.Position1) AND NOT (fb_0.Position2)) AND NOT (fb_0.Position3)));
	testState_0 := testState_0 + 1;
6:
	fb_0.Activate := TRUE; fb_0.S_SafetyActive := TRUE; fb_0.S_FootSwitchCh1 := TRUE; fb_0.S_FootSwitchCh2 := TRUE; fb_0.S_AutoReset := FALSE; fb_0.Reset := FALSE;
	fb_0();
	failed_0 := NOT ((((((((((fb_0.Ready AND fb_0.S_FootSwitchOut) AND fb_0.SafetyDemand) AND NOT (fb_0.ResetRequest)) AND NOT (fb_0.Error)) AND (fb_0.DiagCode = 32768)) AND NOT (fb_0.Reset_Before)) AND NOT (fb_0.Position1)) AND fb_0.Position2) AND NOT (fb_0.Position3)));
	testState_0 := testState_0 + 1;
7:
	fb_0.Activate := TRUE; fb_0.S_SafetyActive := TRUE; fb_0.S_FootSwitchCh1 := TRUE; fb_0.S_FootSwitchCh2 := TRUE; fb_0.S_AutoReset := FALSE; fb_0.Reset := FALSE;
	fb_0();
	failed_0 := NOT ((((((((((fb_0.Ready AND fb_0.S_FootSwitchOut) AND fb_0.SafetyDemand) AND NOT (fb_0.ResetRequest)) AND NOT (fb_0.Error)) AND (fb_0.DiagCode = 32768)) AND NOT (fb_0.Reset_Before)) AND NOT (fb_0.Position1)) AND fb_0.Position2) AND NOT (fb_0.Position3)));
	testState_0 := testState_0 + 1;
8:
	fb_0.Activate := TRUE; fb_0.S_SafetyActive := TRUE; fb_0.S_FootSwitchCh1 := FALSE; fb_0.S_FootSwitchCh2 := TRUE; fb_0.S_AutoReset := FALSE; fb_0.Reset := FALSE;
	fb_0();
	failed_0 := NOT ((((((((((fb_0.Ready AND NOT (fb_0.S_FootSwitchOut)) AND fb_0.SafetyDemand) AND NOT (fb_0.ResetRequest)) AND NOT (fb_0.Error)) AND (fb_0.DiagCode = 32774)) AND NOT (fb_0.Reset_Before)) AND fb_0.Position1) AND NOT (fb_0.Position2)) AND NOT (fb_0.Position3)));
	testState_0 := testState_0 + 1;
9:
	fb_0.Activate := TRUE; fb_0.S_SafetyActive := FALSE; fb_0.S_FootSwitchCh1 := FALSE; fb_0.S_FootSwitchCh2 := TRUE; fb_0.S_AutoReset := FALSE; fb_0.Reset := FALSE;
	fb_0();
	failed_0 := NOT ((((((((((fb_0.Ready AND NOT (fb_0.S_FootSwitchOut)) AND NOT (fb_0.SafetyDemand)) AND NOT (fb_0.ResetRequest)) AND NOT (fb_0.Error)) AND (fb_0.DiagCode = 32772)) AND NOT (fb_0.Reset_Before)) AND fb_0.Position1) AND NOT (fb_0.Position2)) AND NOT (fb_0.Position3)));
	testState_0 := testState_0 + 1;
10:
	fb_0.Activate := TRUE; fb_0.S_SafetyActive := TRUE; fb_0.S_FootSwitchCh1 := FALSE; fb_0.S_FootSwitchCh2 := TRUE; fb_0.S_AutoReset := FALSE; fb_0.Reset := FALSE;
	fb_0();
	failed_0 := NOT ((((((((((fb_0.Ready AND NOT (fb_0.S_FootSwitchOut)) AND NOT (fb_0.SafetyDemand)) AND NOT (fb_0.ResetRequest)) AND NOT (fb_0.Error)) AND (fb_0.DiagCode = 32773)) AND NOT (fb_0.Reset_Before)) AND fb_0.Position1) AND NOT (fb_0.Position2)) AND NOT (fb_0.Position3)));
	testState_0 := testState_0 + 1;
11:
	fb_0.Activate := TRUE; fb_0.S_SafetyActive := TRUE; fb_0.S_FootSwitchCh1 := TRUE; fb_0.S_FootSwitchCh2 := TRUE; fb_0.S_AutoReset := FALSE; fb_0.Reset := FALSE;
	fb_0();
	failed_0 := NOT ((((((((((fb_0.Ready AND NOT (fb_0.S_FootSwitchOut)) AND NOT (fb_0.SafetyDemand)) AND NOT (fb_0.ResetRequest)) AND fb_0.Error) AND (fb_0.DiagCode = 49440)) AND NOT (fb_0.Reset_Before)) AND NOT (fb_0.Position1)) AND fb_0.Position2) AND NOT (fb_0.Position3)));
	testState_0 := testState_0 + 1;
12:
	fb_0.Activate := TRUE; fb_0.S_SafetyActive := TRUE; fb_0.S_FootSwitchCh1 := TRUE; fb_0.S_FootSwitchCh2 := TRUE; fb_0.S_AutoReset := FALSE; fb_0.Reset := FALSE;
	fb_0();
	failed_0 := NOT ((((((((((fb_0.Ready AND NOT (fb_0.S_FootSwitchOut)) AND NOT (fb_0.SafetyDemand)) AND NOT (fb_0.ResetRequest)) AND fb_0.Error) AND (fb_0.DiagCode = 49440)) AND NOT (fb_0.Reset_Before)) AND NOT (fb_0.Position1)) AND fb_0.Position2) AND NOT (fb_0.Position3)));
	testState_0 := testState_0 + 1;
13:
	fb_0.Activate := TRUE; fb_0.S_SafetyActive := TRUE; fb_0.S_FootSwitchCh1 := FALSE; fb_0.S_FootSwitchCh2 := TRUE; fb_0.S_AutoReset := FALSE; fb_0.Reset := TRUE;
	fb_0();
	failed_0 := NOT ((((((((((fb_0.Ready AND NOT (fb_0.S_FootSwitchOut)) AND NOT (fb_0.SafetyDemand)) AND NOT (fb_0.ResetRequest)) AND fb_0.Error) AND (fb_0.DiagCode = 49472)) AND fb_0.Reset_Before) AND fb_0.Position1) AND NOT (fb_0.Position2)) AND NOT (fb_0.Position3)));
	testState_0 := testState_0 + 1;
14:
	fb_0.Activate := TRUE; fb_0.S_SafetyActive := TRUE; fb_0.S_FootSwitchCh1 := FALSE; fb_0.S_FootSwitchCh2 := TRUE; fb_0.S_AutoReset := FALSE; fb_0.Reset := TRUE;
	fb_0();
	failed_0 := NOT ((((((((((fb_0.Ready AND NOT (fb_0.S_FootSwitchOut)) AND NOT (fb_0.SafetyDemand)) AND NOT (fb_0.ResetRequest)) AND fb_0.Error) AND (fb_0.DiagCode = 49473)) AND fb_0.Reset_Before) AND fb_0.Position1) AND NOT (fb_0.Position2)) AND NOT (fb_0.Position3)));
	testState_0 := testState_0 + 1;
15:
	fb_0.Activate := TRUE; fb_0.S_SafetyActive := TRUE; fb_0.S_FootSwitchCh1 := FALSE; fb_0.S_FootSwitchCh2 := TRUE; fb_0.S_AutoReset := FALSE; fb_0.Reset := TRUE;
	fb_0();
	failed_0 := NOT ((((((((((fb_0.Ready AND NOT (fb_0.S_FootSwitchOut)) AND NOT (fb_0.SafetyDemand)) AND NOT (fb_0.ResetRequest)) AND fb_0.Error) AND (fb_0.DiagCode = 49473)) AND fb_0.Reset_Before) AND fb_0.Position1) AND NOT (fb_0.Position2)) AND NOT (fb_0.Position3)));
	testState_0 := testState_0 + 1;
16:
	fb_0.Activate := TRUE; fb_0.S_SafetyActive := TRUE; fb_0.S_FootSwitchCh1 := FALSE; fb_0.S_FootSwitchCh2 := TRUE; fb_0.S_AutoReset := FALSE; fb_0.Reset := FALSE;
	fb_0();
	failed_0 := NOT ((((((((((fb_0.Ready AND NOT (fb_0.S_FootSwitchOut)) AND NOT (fb_0.SafetyDemand)) AND NOT (fb_0.ResetRequest)) AND fb_0.Error) AND (fb_0.DiagCode = 49472)) AND NOT (fb_0.Reset_Before)) AND fb_0.Position1) AND NOT (fb_0.Position2)) AND NOT (fb_0.Position3)));
	testState_0 := testState_0 + 1;
17:
	fb_0.Activate := TRUE; fb_0.S_SafetyActive := TRUE; fb_0.S_FootSwitchCh1 := FALSE; fb_0.S_FootSwitchCh2 := TRUE; fb_0.S_AutoReset := FALSE; fb_0.Reset := FALSE;
	fb_0();
	failed_0 := NOT ((((((((((fb_0.Ready AND NOT (fb_0.S_FootSwitchOut)) AND NOT (fb_0.SafetyDemand)) AND NOT (fb_0.ResetRequest)) AND fb_0.Error) AND (fb_0.DiagCode = 49472)) AND NOT (fb_0.Reset_Before)) AND fb_0.Position1) AND NOT (fb_0.Position2)) AND NOT (fb_0.Position3)));
	testState_0 := testState_0 + 1;
18:
	fb_0.Activate := TRUE; fb_0.S_SafetyActive := TRUE; fb_0.S_FootSwitchCh1 := TRUE; fb_0.S_FootSwitchCh2 := TRUE; fb_0.S_AutoReset := FALSE; fb_0.Reset := FALSE;
	fb_0();
	failed_0 := NOT ((((((((((fb_0.Ready AND NOT (fb_0.S_FootSwitchOut)) AND NOT (fb_0.SafetyDemand)) AND NOT (fb_0.ResetRequest)) AND fb_0.Error) AND (fb_0.DiagCode = 49440)) AND NOT (fb_0.Reset_Before)) AND NOT (fb_0.Position1)) AND fb_0.Position2) AND NOT (fb_0.Position3)));
	testState_0 := testState_0 + 1;
19:
	fb_0.Activate := TRUE; fb_0.S_SafetyActive := TRUE; fb_0.S_FootSwitchCh1 := FALSE; fb_0.S_FootSwitchCh2 := TRUE; fb_0.S_AutoReset := FALSE; fb_0.Reset := FALSE;
	fb_0();
	failed_0 := NOT ((((((((((fb_0.Ready AND NOT (fb_0.S_FootSwitchOut)) AND NOT (fb_0.SafetyDemand)) AND NOT (fb_0.ResetRequest)) AND fb_0.Error) AND (fb_0.DiagCode = 49472)) AND NOT (fb_0.Reset_Before)) AND fb_0.Position1) AND NOT (fb_0.Position2)) AND NOT (fb_0.Position3)));
	testState_0 := testState_0 + 1;
20:
	fb_0.Activate := TRUE; fb_0.S_SafetyActive := TRUE; fb_0.S_FootSwitchCh1 := FALSE; fb_0.S_FootSwitchCh2 := TRUE; fb_0.S_AutoReset := FALSE; fb_0.Reset := TRUE;
	fb_0();
	failed_0 := NOT ((((((((((fb_0.Ready AND NOT (fb_0.S_FootSwitchOut)) AND fb_0.SafetyDemand) AND NOT (fb_0.ResetRequest)) AND NOT (fb_0.Error)) AND (fb_0.DiagCode = 32774)) AND fb_0.Reset_Before) AND fb_0.Position1) AND NOT (fb_0.Position2)) AND NOT (fb_0.Position3)));
	testState_0 := testState_0 + 1;
21:
	fb_0.Activate := TRUE; fb_0.S_SafetyActive := TRUE; fb_0.S_FootSwitchCh1 := FALSE; fb_0.S_FootSwitchCh2 := FALSE; fb_0.S_AutoReset := FALSE; fb_0.Reset := FALSE;
	fb_0();
	failed_0 := NOT ((((((((((fb_0.Ready AND NOT (fb_0.S_FootSwitchOut)) AND fb_0.SafetyDemand) AND NOT (fb_0.ResetRequest)) AND NOT (fb_0.Error)) AND (fb_0.DiagCode = 34832)) AND NOT (fb_0.Reset_Before)) AND NOT (fb_0.Position1)) AND NOT (fb_0.Position2)) AND fb_0.Position3));
	testState_0 := testState_0 + 1;
22:
	fb_0.Activate := TRUE; fb_0.S_SafetyActive := TRUE; fb_0.S_FootSwitchCh1 := TRUE; fb_0.S_FootSwitchCh2 := FALSE; fb_0.S_AutoReset := FALSE; fb_0.Reset := FALSE;
	fb_0();
	failed_0 := NOT ((((((((((fb_0.Ready AND NOT (fb_0.S_FootSwitchOut)) AND fb_0.SafetyDemand) AND NOT (fb_0.ResetRequest)) AND NOT (fb_0.Error)) AND (fb_0.DiagCode = 34832)) AND NOT (fb_0.Reset_Before)) AND NOT (fb_0.Position1)) AND NOT (fb_0.Position2)) AND fb_0.Position3));
	testState_0 := testState_0 + 1;
23:
	fb_0.Activate := TRUE; fb_0.S_SafetyActive := TRUE; fb_0.S_FootSwitchCh1 := FALSE; fb_0.S_FootSwitchCh2 := TRUE; fb_0.S_AutoReset := FALSE; fb_0.Reset := FALSE;
	fb_0();
	failed_0 := NOT ((((((((((fb_0.Ready AND NOT (fb_0.S_FootSwitchOut)) AND fb_0.SafetyDemand) AND NOT (fb_0.ResetRequest)) AND NOT (fb_0.Error)) AND (fb_0.DiagCode = 32774)) AND NOT (fb_0.Reset_Before)) AND fb_0.Position1) AND NOT (fb_0.Position2)) AND NOT (fb_0.Position3)));
	testState_0 := testState_0 + 1;
24:
	fb_0.Activate := TRUE; fb_0.S_SafetyActive := TRUE; fb_0.S_FootSwitchCh1 := TRUE; fb_0.S_FootSwitchCh2 := TRUE; fb_0.S_AutoReset := FALSE; fb_0.Reset := FALSE;
	fb_0();
	failed_0 := NOT ((((((((((fb_0.Ready AND fb_0.S_FootSwitchOut) AND fb_0.SafetyDemand) AND NOT (fb_0.ResetRequest)) AND NOT (fb_0.Error)) AND (fb_0.DiagCode = 32768)) AND NOT (fb_0.Reset_Before)) AND NOT (fb_0.Position1)) AND fb_0.Position2) AND NOT (fb_0.Position3)));
	testState_0 := testState_0 + 1;
25:
	fb_0.Activate := TRUE; fb_0.S_SafetyActive := TRUE; fb_0.S_FootSwitchCh1 := FALSE; fb_0.S_FootSwitchCh2 := FALSE; fb_0.S_AutoReset := FALSE; fb_0.Reset := FALSE;
	fb_0();
	failed_0 := NOT ((((((((((fb_0.Ready AND NOT (fb_0.S_FootSwitchOut)) AND fb_0.SafetyDemand) AND NOT (fb_0.ResetRequest)) AND NOT (fb_0.Error)) AND (fb_0.DiagCode = 34832)) AND NOT (fb_0.Reset_Before)) AND NOT (fb_0.Position1)) AND NOT (fb_0.Position2)) AND fb_0.Position3));
	testState_0 := testState_0 + 1;
26:
	fb_0.Activate := TRUE; fb_0.S_SafetyActive := TRUE; fb_0.S_FootSwitchCh1 := TRUE; fb_0.S_FootSwitchCh2 := TRUE; fb_0.S_AutoReset := FALSE; fb_0.Reset := FALSE;
	fb_0();
	failed_0 := NOT ((((((((((fb_0.Ready AND NOT (fb_0.S_FootSwitchOut)) AND NOT (fb_0.SafetyDemand)) AND NOT (fb_0.ResetRequest)) AND fb_0.Error) AND (fb_0.DiagCode = 49504)) AND NOT (fb_0.Reset_Before)) AND NOT (fb_0.Position1)) AND fb_0.Position2) AND NOT (fb_0.Position3)));
	testState_0 := testState_0 + 1;
27:
	fb_0.Activate := TRUE; fb_0.S_SafetyActive := TRUE; fb_0.S_FootSwitchCh1 := TRUE; fb_0.S_FootSwitchCh2 := TRUE; fb_0.S_AutoReset := FALSE; fb_0.Reset := FALSE;
	fb_0();
	failed_0 := NOT ((((((((((fb_0.Ready AND NOT (fb_0.S_FootSwitchOut)) AND NOT (fb_0.SafetyDemand)) AND NOT (fb_0.ResetRequest)) AND fb_0.Error) AND (fb_0.DiagCode = 49504)) AND NOT (fb_0.Reset_Before)) AND NOT (fb_0.Position1)) AND fb_0.Position2) AND NOT (fb_0.Position3)));
	testState_0 := testState_0 + 1;
28:
	fb_0.Activate := TRUE; fb_0.S_SafetyActive := TRUE; fb_0.S_FootSwitchCh1 := FALSE; fb_0.S_FootSwitchCh2 := TRUE; fb_0.S_AutoReset := FALSE; fb_0.Reset := TRUE;
	fb_0();
	failed_0 := NOT ((((((((((fb_0.Ready AND NOT (fb_0.S_FootSwitchOut)) AND NOT (fb_0.SafetyDemand)) AND NOT (fb_0.ResetRequest)) AND fb_0.Error) AND (fb_0.DiagCode = 49536)) AND fb_0.Reset_Before) AND fb_0.Position1) AND NOT (fb_0.Position2)) AND NOT (fb_0.Position3)));
	testState_0 := testState_0 + 1;
29:
	fb_0.Activate := TRUE; fb_0.S_SafetyActive := TRUE; fb_0.S_FootSwitchCh1 := FALSE; fb_0.S_FootSwitchCh2 := TRUE; fb_0.S_AutoReset := FALSE; fb_0.Reset := TRUE;
	fb_0();
	failed_0 := NOT ((((((((((fb_0.Ready AND NOT (fb_0.S_FootSwitchOut)) AND NOT (fb_0.SafetyDemand)) AND NOT (fb_0.ResetRequest)) AND fb_0.Error) AND (fb_0.DiagCode = 49537)) AND fb_0.Reset_Before) AND fb_0.Position1) AND NOT (fb_0.Position2)) AND NOT (fb_0.Position3)));
	testState_0 := testState_0 + 1;
30:
	fb_0.Activate := TRUE; fb_0.S_SafetyActive := TRUE; fb_0.S_FootSwitchCh1 := FALSE; fb_0.S_FootSwitchCh2 := TRUE; fb_0.S_AutoReset := FALSE; fb_0.Reset := TRUE;
	fb_0();
	failed_0 := NOT ((((((((((fb_0.Ready AND NOT (fb_0.S_FootSwitchOut)) AND NOT (fb_0.SafetyDemand)) AND NOT (fb_0.ResetRequest)) AND fb_0.Error) AND (fb_0.DiagCode = 49537)) AND fb_0.Reset_Before) AND fb_0.Position1) AND NOT (fb_0.Position2)) AND NOT (fb_0.Position3)));
	testState_0 := testState_0 + 1;
31:
	fb_0.Activate := TRUE; fb_0.S_SafetyActive := TRUE; fb_0.S_FootSwitchCh1 := FALSE; fb_0.S_FootSwitchCh2 := TRUE; fb_0.S_AutoReset := FALSE; fb_0.Reset := FALSE;
	fb_0();
	failed_0 := NOT ((((((((((fb_0.Ready AND NOT (fb_0.S_FootSwitchOut)) AND NOT (fb_0.SafetyDemand)) AND NOT (fb_0.ResetRequest)) AND fb_0.Error) AND (fb_0.DiagCode = 49536)) AND NOT (fb_0.Reset_Before)) AND fb_0.Position1) AND NOT (fb_0.Position2)) AND NOT (fb_0.Position3)));
	testState_0 := testState_0 + 1;
32:
	fb_0.Activate := TRUE; fb_0.S_SafetyActive := TRUE; fb_0.S_FootSwitchCh1 := FALSE; fb_0.S_FootSwitchCh2 := TRUE; fb_0.S_AutoReset := FALSE; fb_0.Reset := FALSE;
	fb_0();
	failed_0 := NOT ((((((((((fb_0.Ready AND NOT (fb_0.S_FootSwitchOut)) AND NOT (fb_0.SafetyDemand)) AND NOT (fb_0.ResetRequest)) AND fb_0.Error) AND (fb_0.DiagCode = 49536)) AND NOT (fb_0.Reset_Before)) AND fb_0.Position1) AND NOT (fb_0.Position2)) AND NOT (fb_0.Position3)));
	testState_0 := testState_0 + 1;
33:
	fb_0.Activate := TRUE; fb_0.S_SafetyActive := TRUE; fb_0.S_FootSwitchCh1 := TRUE; fb_0.S_FootSwitchCh2 := TRUE; fb_0.S_AutoReset := FALSE; fb_0.Reset := FALSE;
	fb_0();
	failed_0 := NOT ((((((((((fb_0.Ready AND NOT (fb_0.S_FootSwitchOut)) AND NOT (fb_0.SafetyDemand)) AND NOT (fb_0.ResetRequest)) AND fb_0.Error) AND (fb_0.DiagCode = 49504)) AND NOT (fb_0.Reset_Before)) AND NOT (fb_0.Position1)) AND fb_0.Position2) AND NOT (fb_0.Position3)));
	testState_0 := testState_0 + 1;
34:
	fb_0.Activate := TRUE; fb_0.S_SafetyActive := TRUE; fb_0.S_FootSwitchCh1 := FALSE; fb_0.S_FootSwitchCh2 := TRUE; fb_0.S_AutoReset := FALSE; fb_0.Reset := FALSE;
	fb_0();
	failed_0 := NOT ((((((((((fb_0.Ready AND NOT (fb_0.S_FootSwitchOut)) AND NOT (fb_0.SafetyDemand)) AND NOT (fb_0.ResetRequest)) AND fb_0.Error) AND (fb_0.DiagCode = 49536)) AND NOT (fb_0.Reset_Before)) AND fb_0.Position1) AND NOT (fb_0.Position2)) AND NOT (fb_0.Position3)));
	testState_0 := testState_0 + 1;
35:
	fb_0.Activate := TRUE; fb_0.S_SafetyActive := TRUE; fb_0.S_FootSwitchCh1 := FALSE; fb_0.S_FootSwitchCh2 := FALSE; fb_0.S_AutoReset := FALSE; fb_0.Reset := TRUE;
	fb_0();
	failed_0 := NOT ((((((((((fb_0.Ready AND NOT (fb_0.S_FootSwitchOut)) AND fb_0.SafetyDemand) AND NOT (fb_0.ResetRequest)) AND NOT (fb_0.Error)) AND (fb_0.DiagCode = 34832)) AND fb_0.Reset_Before) AND NOT (fb_0.Position1)) AND NOT (fb_0.Position2)) AND fb_0.Position3));
	testState_0 := testState_0 + 1;
36:
	fb_0.Activate := TRUE; fb_0.S_SafetyActive := FALSE; fb_0.S_FootSwitchCh1 := FALSE; fb_0.S_FootSwitchCh2 := TRUE; fb_0.S_AutoReset := FALSE; fb_0.Reset := FALSE;
	fb_0();
	failed_0 := NOT ((fb_0.Ready AND (NOT (fb_0.S_FootSwitchOut) AND (NOT (fb_0.SafetyDemand) AND (NOT (fb_0.ResetRequest) AND (NOT (fb_0.Error) AND ((fb_0.DiagCode = 32772) AND (NOT (fb_0.Reset_Before) AND (NOT (fb_0.Position1) AND (NOT (fb_0.Position2) AND fb_0.Position3))))))))));
	testState_0 := testState_0 + 1;
37:
	finished_0 := TRUE;
END_CASE
END_IF

END_FUNCTION_BLOCK

(* ---- SF_ModeSelector.st ---- *)
FUNCTION_BLOCK SF_ModeSelector
VAR_INPUT
    Activate: BOOL;
    S_Mode0: BOOL;
    S_Mode1: BOOL;
    S_Mode2: BOOL;
    S_Mode3: BOOL;
    S_Mode4: BOOL;
    S_Mode5: BOOL;
    S_Mode6: BOOL;
    S_Mode7: BOOL;
    AutoSetMode: BOOL;
    S_SetMode: BOOL;
    S_Unlock: BOOL;
    Reset: BOOL;
    ModeMonitorTime: TIME := T#100MS;
END_VAR
VAR_OUTPUT
    Ready: BOOL;
    S_Mode0Sel: BOOL;
    S_Mode1Sel: BOOL;
    S_Mode2Sel: BOOL;
    S_Mode3Sel: BOOL;
    S_Mode4Sel: BOOL;
    S_Mode5Sel: BOOL;
    S_Mode6Sel: BOOL;
    S_Mode7Sel: BOOL;
    S_AnyModeSel: BOOL;
    SafetyDemand: BOOL;
    ResetRequest: BOOL;
    Error: BOOL;
    DiagCode: UINT;
END_VAR
VAR
    T_1: TON;
    Reset_Before: BOOL;
    S_SetMode_Before: BOOL;
END_VAR

VAR_TEMP
    ModeSum: USINT;
    ModeChanged: BOOL;
    Error1: BOOL;
    Error2: BOOL;
END_VAR

BEGIN

IF NOT Activate THEN
    DiagCode := 16#0000;

    Ready := FALSE;
    SafetyDemand := FALSE;
    ResetRequest := FALSE;
    Error := FALSE;
    S_AnyModeSel := FALSE;
    S_Mode0Sel := FALSE;
    S_Mode1Sel := FALSE;
    S_Mode2Sel := FALSE;
    S_Mode3Sel := FALSE;
    S_Mode4Sel := FALSE;
    S_Mode5Sel := FALSE;
    S_Mode6Sel := FALSE;
    S_Mode7Sel := FALSE;

    T_1(IN := 0);
    Reset_Before := FALSE;
    S_SetMode_Before := FALSE;

    ModeSum := 0;
    ModeChanged := FALSE;
    Error1 := FALSE;
    Error2 := FALSE;
ELSE
    T_1(PT := ModeMonitorTime);

    ModeSum := 0;
    IF S_Mode0 THEN
        ModeSum := ModeSum+1;
    END_IF;
    IF S_Mode1 THEN
        ModeSum := ModeSum+1;
    END_IF;
    IF S_Mode2 THEN
        ModeSum := ModeSum+1;
    END_IF;
    IF S_Mode3 THEN
        ModeSum := ModeSum+1;
    END_IF;
    IF S_Mode4 THEN
        ModeSum := ModeSum+1;
    END_IF;
    IF S_Mode5 THEN
        ModeSum := ModeSum+1;
    END_IF;
    IF S_Mode6 THEN
        ModeSum := ModeSum+1;
    END_IF;
    IF S_Mode7 THEN
        ModeSum := ModeSum+1;
    END_IF;

    IF S_Mode0 <> S_Mode0Sel THEN
        ModeChanged := TRUE;
    ELSIF S_Mode1 <> S_Mode1Sel THEN
        ModeChanged := TRUE;
    ELSIF S_Mode2 <> S_Mode2Sel THEN
        ModeChanged := TRUE;
    ELSIF S_Mode3 <> S_Mode3Sel THEN
        ModeChanged := TRUE;
    ELSIF S_Mode4 <> S_Mode4Sel THEN
        ModeChanged := TRUE;
    ELSIF S_Mode5 <> S_Mode5Sel THEN
        ModeChanged := TRUE;
    ELSIF S_Mode6 <> S_Mode6Sel THEN
        ModeChanged := TRUE;
    ELSIF S_Mode7 <> S_Mode7Sel THEN
        ModeChanged := TRUE;
    ELSE
        ModeChanged := FALSE;
    END_IF;

    IF ModeSum > 1 THEN
        Error1 := true;
    ELSE
        Error1 := false;
    END_IF;

    // state changes
    CASE DiagCode OF
    16#0000:
        DiagCode := 16#8802;
        T_1(IN := 0);
        T_1(IN := 1, PT := ModeMonitorTime);
    16#8802:
        IF Error1 THEN
            T_1(IN := 0);
            DiagCode := 16#C010;
        ELSIF T_1.Q THEN
            DiagCode := 16#C020;
        ELSIF (AutoSetMode OR (NOT S_SetMode_Before AND S_SetMode)) AND S_Unlock AND (ModeSum = 1) THEN
            T_1(IN := 0);
            DiagCode := 16#8000;
            S_Mode0Sel := S_Mode0;
            S_Mode1Sel := S_Mode1;
            S_Mode2Sel := S_Mode2;
            S_Mode3Sel := S_Mode3;
            S_Mode4Sel := S_Mode4;
            S_Mode5Sel := S_Mode5;
            S_Mode6Sel := S_Mode6;
            S_Mode7Sel := S_Mode7;
        END_IF;
    16#8000:
        IF Error1 THEN
            DiagCode := 16#C010;
        ELSIF ModeChanged THEN
            DiagCode := 16#8802;
            T_1(IN := 0);
            T_1(IN := 1, PT := ModeMonitorTime);
        ELSIF NOT S_Unlock THEN
            DiagCode := 16#8010;
        END_IF;
    16#8010:
        IF S_Unlock THEN
            IF Error1 THEN
                DiagCode := 16#C010;
            ELSIF ModeChanged THEN
                DiagCode := 16#8802;
                T_1(IN := 0);
                T_1(IN := 1, PT := ModeMonitorTime);
            ELSE
                DiagCode := 16#8000;
            END_IF;
        END_IF;
    16#C010:
        IF Reset_Before AND Reset THEN
            DiagCode := 16#C011;
        ELSIF (ModeSum = 0) OR (ModeSum = 1) THEN
            IF NOT Reset_Before AND Reset THEN
                DiagCode := 16#8802;
                T_1(IN := 0);
                T_1(IN := 1, PT := ModeMonitorTime);
            ELSE
                DiagCode := 16#C410;
            END_IF;
        END_IF;
    16#C410:
        IF Reset_Before AND Reset THEN
            DiagCode := 16#C011;
        ELSIF (ModeSum = 0) OR (ModeSum = 1) THEN
            IF NOT Reset_Before AND Reset THEN
                DiagCode := 16#8802;
                T_1(IN := 0);
                T_1(IN := 1, PT := ModeMonitorTime);
            END_IF;
        ELSE
            DiagCode := 16#C010;
        END_IF;
    16#C020:
        IF Reset_Before AND Reset THEN
            DiagCode := 16#C021;
        ELSIF (ModeSum = 1) THEN
            IF NOT Reset_Before AND Reset THEN
                DiagCode := 16#8802;
                T_1(IN := 0);
                T_1(IN := 1, PT := ModeMonitorTime);
            ELSE
                DiagCode := 16#C420;
            END_IF;
        END_IF;
    16#C420:
        IF Reset_Before AND Reset THEN
            DiagCode := 16#C021;
        ELSIF (ModeSum = 1) THEN
            IF NOT Reset_Before AND Reset THEN
                DiagCode := 16#8802;
                T_1(IN := 0);
                T_1(IN := 1, PT := ModeMonitorTime);
            END_IF;
        ELSE
            DiagCode := 16#C020;
        END_IF;
    16#C011:
        IF (NOT Reset) THEN
            DiagCode := 16#C010;
        END_IF;
    16#C021:
        IF (NOT Reset) THEN
            DiagCode := 16#C020;
        END_IF;
    END_CASE;

    // set output variables
    CASE DiagCode OF
    16#8802:
        Ready := TRUE;
        SafetyDemand := TRUE;
        ResetRequest := FALSE;
        Error := FALSE;
        S_AnyModeSel := FALSE;
        S_Mode0Sel := FALSE;
        S_Mode1Sel := FALSE;
        S_Mode2Sel := FALSE;
        S_Mode3Sel := FALSE;
        S_Mode4Sel := FALSE;
        S_Mode5Sel := FALSE;
        S_Mode6Sel := FALSE;
        S_Mode7Sel := FALSE;
    16#8000:
        Ready := TRUE;
        SafetyDemand := FALSE;
        ResetRequest := FALSE;
        Error := FALSE;
        S_AnyModeSel := TRUE;
    16#8010:
        Ready := TRUE;
        SafetyDemand := FALSE;
        ResetRequest := FALSE;
        Error := FALSE;
        S_AnyModeSel := TRUE;
    16#C010:
        Ready := TRUE;
        SafetyDemand := FALSE;
        ResetRequest := FALSE;
        Error := TRUE;
        S_AnyModeSel := FALSE;
        S_Mode0Sel := FALSE;
        S_Mode1Sel := FALSE;
        S_Mode2Sel := FALSE;
        S_Mode3Sel := FALSE;
        S_Mode4Sel := FALSE;
        S_Mode5Sel := FALSE;
        S_Mode6Sel := FALSE;
        S_Mode7Sel := FALSE;
    16#C410:
        Ready := TRUE;
        SafetyDemand := FALSE;
        ResetRequest := NOT Reset;
        Error := TRUE;
        S_AnyModeSel := FALSE;
        S_Mode0Sel := FALSE;
        S_Mode1Sel := FALSE;
        S_Mode2Sel := FALSE;
        S_Mode3Sel := FALSE;
        S_Mode4Sel := FALSE;
        S_Mode5Sel := FALSE;
        S_Mode6Sel := FALSE;
        S_Mode7Sel := FALSE;
    16#C020:
        Ready := TRUE;
        SafetyDemand := FALSE;
        ResetRequest := FALSE;
        Error := TRUE;
        S_AnyModeSel := FALSE;
        S_Mode0Sel := FALSE;
        S_Mode1Sel := FALSE;
        S_Mode2Sel := FALSE;
        S_Mode3Sel := FALSE;
        S_Mode4Sel := FALSE;
        S_Mode5Sel := FALSE;
        S_Mode6Sel := FALSE;
        S_Mode7Sel := FALSE;
    16#C420:
        Ready := TRUE;
        SafetyDemand := FALSE;
        ResetRequest := NOT Reset;
        Error := TRUE;
        S_AnyModeSel := FALSE;
        S_Mode0Sel := FALSE;
        S_Mode1Sel := FALSE;
        S_Mode2Sel := FALSE;
        S_Mode3Sel := FALSE;
        S_Mode4Sel := FALSE;
        S_Mode5Sel := FALSE;
        S_Mode6Sel := FALSE;
        S_Mode7Sel := FALSE;
    16#C011:
        Ready := TRUE;
        SafetyDemand := FALSE;
        ResetRequest := FALSE;
        Error := TRUE;
        S_AnyModeSel := FALSE;
        S_Mode0Sel := FALSE;
        S_Mode1Sel := FALSE;
        S_Mode2Sel := FALSE;
        S_Mode3Sel := FALSE;
        S_Mode4Sel := FALSE;
        S_Mode5Sel := FALSE;
        S_Mode6Sel := FALSE;
        S_Mode7Sel := FALSE;
    16#C021:
        Ready := TRUE;
        SafetyDemand := FALSE;
        ResetRequest := FALSE;
        Error := TRUE;
        S_AnyModeSel := FALSE;
        S_Mode0Sel := FALSE;
        S_Mode1Sel := FALSE;
        S_Mode2Sel := FALSE;
        S_Mode3Sel := FALSE;
        S_Mode4Sel := FALSE;
        S_Mode5Sel := FALSE;
        S_Mode6Sel := FALSE;
        S_Mode7Sel := FALSE;
    END_CASE;

    Reset_Before := Reset;
    S_SetMode_Before := S_SetMode;
END_IF;

END_FUNCTION_BLOCK
